Fanuc KAREL source: kb00016.KL

-- PROVISIONAL review KL for V770-1; original PC SHA256 2749ca15c896e337036673263026a6d65ab9c112a18dea1bfc640f42b0bf9066
-- Incomplete behavior may be omitted. Consult companion uncertainty JSON. Do not deploy.
PROGRAM KB00016
%NOLOCKGROUP
BEGIN
  -- UNRESOLVED_PC offsets 5-14; opcodes 3F,75
  -- UNRESOLVED_PC offsets 19-26; opcodes 9D,23
  -- UNRESOLVED_PC offsets 31-38; opcodes 9D,23
  -- UNRESOLVED_PC offsets 43-50; opcodes 9D,23
  -- UNRESOLVED_PC offsets 55-85; opcodes 27,22,2A,22,22,22,31
  -- UNRESOLVED_PC offsets 90-94; opcodes 7F
END KB00016
